FUNCTION_BLOCK TestFileLogger EXTENDS TcUnit.FB_TestSuite
VAR_INPUT
END_VAR
VAR_OUTPUT
END_VAR
VAR
END_VAR

END_FUNCTION_BLOCK

(* stored: Version 1.1.0.1, ProductVersion 3.1.4022.18
   POU TestFileLogger: Id {6eb9b79c-7996-4180-884f-6c85712e4467}, SpecialFunc None *)
